(* PLC project Generated_UR10eControl, CODESYS CODESYS V3.5 SP20 Patch 3 *)
(* stored: creationDateTime 2026-01-30T19:43:14.0000000, modificationDateTime 2026-01-30T19:43:14.0000000 *)

TYPE ST_UR10eControl : STRUCT
  ToCPP : ST_ToCPP;
  FromCPP : ST_FromCPP;
  LifePLC : DINT;  (* PLC heartbeat counter *)
  LifeCPP : DINT;  (* C++ heartbeat counter *)
END_STRUCT;
END_TYPE

TYPE ST_ToCPP : STRUCT
  shoulder_pan_joint : LREAL;
  shoulder_lift_joint : LREAL;
  elbow_joint : LREAL;
  wrist_1_joint : LREAL;
  wrist_2_joint : LREAL;
  wrist_3_joint : LREAL;
END_STRUCT;
END_TYPE

TYPE ST_FromCPP : STRUCT
  shoulder_pan_joint_sensor : LREAL;
  shoulder_lift_joint_sensor : LREAL;
  elbow_joint_sensor : LREAL;
  wrist_1_joint_sensor : LREAL;
  wrist_2_joint_sensor : LREAL;
  wrist_3_joint_sensor : LREAL;
END_STRUCT;
END_TYPE
